// TIA Portal V17 export
// export: Created 2025-03-10T13:12:15.8739862Z, ExportSetting WithDefaults, DisplayName Totally Integrated Automation Portal, DisplayVersion V17 Update 8, DisplayName TIA Portal Openness, DisplayVersion V17 Update 8, DisplayName TIA Portal Version Control Interface, DisplayVersion V17, DisplayName SINAMICS Startdrive Advanced, DisplayVersion V17 SP2, DisplayName SINAMICS Startdrive G110M, G120, G120C, G120D, G120P, G115D, DisplayVersion V17 SP2, DisplayName SINAMICS Startdrive G130, G150, S120, S150, SINAMICS MV, S210, DisplayVersion V17 SP2, DisplayName STEP 7 Professional, DisplayVersion V17 Update 8, DisplayName SINUMERIK ONE STEP 7 Toolbox, DisplayVersion V17 Update 12, DisplayName SINUMERIK 840D sl STEP 7 Toolbox, DisplayVersion V17 Update 12, DisplayName STEP 7 Safety, DisplayVersion V17 Update 6, DisplayName WinCC Advanced, DisplayVersion V17 Update 8
TYPE "READ_CNC_MEMORY_2"
// stored: IsFailsafeCompliant false
   STRUCT
      Index : Word;   // Index, 1 = Arbeitsspeicher
      Code : Word;   // Speichertyp, 1 = RAM, 2 = FEPROM, 3 = RAM und FEPROM
      Size : DWord;   // Gesamtgroesse
      Mode : Word;   // Modus, Bit 0=RAM, 1=FEPROM, 2=RAM/FEPROM, 3=Code/Daten getr., 4=Code/Daten gem.
      Granu : Word;   // Immer 0
      Ber1 : DWord;   // Groesse des RAM's
      Occupied1 : DWord;   // Groesse des belegten RAM's
      Block1 : DWord;   // Groesster freier Block
      Ber2 : DWord;   // Groesse des FEPROM's
      Occupied2 : DWord;   // Groesse des belegten FEPROM's
      Block2 : DWord;   // Groesster frreier Block
   END_STRUCT;
END_TYPE
